TYPE REAL2 :
STRUCT
	R1 : REAL;	(* small value *)
	RX : REAL;	(* big value *)
END_STRUCT
END_TYPE

(* stored: Version 1.1.0.1
   DUT REAL2: Id {da7a2ded-2271-4eb6-986a-83f6527d2db3} *)
